PROGRAM MAIN
VAR
	FB_ClkSignal_1	:	FB_ClkSignal;
END_VAR

FB_ClkSignal_1(IN_bStart:= , IN_fFrequency:=0.001 , OUT_Signal=> );

END_PROGRAM

(* stored: Version 1.1.0.1, ProductVersion 3.1.4024.4
   POU MAIN: Id {cfae907d-2971-42a4-b8bc-d377595e7a12}, SpecialFunc None *)
